{attribute 'qualified_only'}
{attribute 'strict'}
TYPE VacuumBeltTableMode :
(
	Mode_Standard	:= 0,
	Mode_Manual		:= 1,
	Mode_Simulation	:= 2
	
);
END_TYPE

(* stored: Version 1.1.0.1, ProductVersion 3.1.4024.12
   DUT VacuumBeltTableMode: Id {454b8484-127c-4d56-8ba5-0bbde54cd307} *)
